// TIA Portal V20 export
TYPE "typeEm6Standard"
// stored: Access Published, Namespace Unit1
   STRUCT
      commands { ExternalWritable := 'False'} : "Unit1.typeEm6Commands";
      monitoring { ExternalWritable := 'False'} : "Unit1.typeEm6Monitoring";
   END_STRUCT;
END_TYPE
